PROGRAM F_FactoryIO_WriteRegs
VAR
	LFB_MBWriteRegs  	: FB_MBWriteRegs ;
	bBusy: BOOL;
	bError: BOOL;

END_VAR

LFB_MBWriteRegs(
	sIPAddr := '127.0.0.1',
	nTCPPort := 505,
	nUnitID := 255,
	nQuantity := 8,
	nMBAddr := 0,
	cbLength := SIZEOF(GAB_FactoryIO_OutputsRegs),
	pSrcAddr:= ADR(GAB_FactoryIO_OutputsRegs), 
	bExecute := TRUE,
	tTimeout := T#1S,
	bBusy=> bBusy, 
	bError=> bError, 
	nErrId=>
);
LFB_MBWriteRegs(bExecute := FALSE);

END_PROGRAM

(* stored: Version 1.1.0.1, ProductVersion 3.1.4024.11
   POU F_FactoryIO_WriteRegs: Id {7b35c821-98cd-42f3-9186-98d8239ea522}, SpecialFunc None *)
